FUNCTION_BLOCK FB_DiagnosisEtherCATMaster
VAR_INPUT
	sMasterName					:STRING	:='NameNotSet';				//マスター名
END_VAR
VAR_IN_OUT
	fbFrmWcStateDiagnosis		:ARRAY[*] OF FB_FrmWcStateDiagnosis;
	fbFrmStateDiagnosis			:ARRAY[*] OF FB_FrmStateDiagnosis;
END_VAR
VAR_OUTPUT
	bError						:BOOL;								//エラー発生を出力
END_VAR
VAR
	fbDevStateDiagnosis			:FB_DevStateDiagnosis;
	fbSlaveCountDiagnosis		:FB_SlaveCountDiagnosis;
	i							:DINT;
END_VAR

//診断用FBを呼び出し
fbDevStateDiagnosis(sMasterName:=sMasterName);
fbSlaveCountDiagnosis(sMasterName:=sMasterName);

bError:=fbDevStateDiagnosis.bError OR fbSlaveCountDiagnosis.bError;

//可変長のアレイを診断と出力
FOR i := LOWER_BOUND(fbFrmWcStateDiagnosis,1) TO UPPER_BOUND(fbFrmWcStateDiagnosis,1) DO
	fbFrmWcStateDiagnosis[i](sMasterName:=sMasterName);
	bError:=bError OR fbFrmWcStateDiagnosis[i].bError;
END_FOR

FOR i := LOWER_BOUND(fbFrmStateDiagnosis,1) TO UPPER_BOUND(fbFrmStateDiagnosis,1) DO
	fbFrmStateDiagnosis[i](sMasterName:=sMasterName);
	bError:=bError OR fbFrmStateDiagnosis[i].bError;
END_FOR

END_FUNCTION_BLOCK

(* stored: Version 1.1.0.1
   POU FB_DiagnosisEtherCATMaster: Id {de43cf2f-fd79-46c9-9b8b-af34aac85cac}, SpecialFunc None *)
